{attribute addProperty BoxType "BK1250-0000-0017"}
{attribute addProperty Id "Term_387_KL1002KL1002_D229A9CA00"}
{attribute addProperty CRC "1147850243"}
{attribute addProperty SizeInBites "0"}
{attribute addProperty SizeInBytes "0"}
TYPE A_0016_BK1250_0000_0017_446ACE03 EXTENDS BK1250_4487A81F :
STRUCT
	{attribute addProperty Name "Term_387_KL1002"}
	Term_387_KL1002 : KL1002_D229A9CA;
END_STRUCT
END_TYPE

(* stored: Version 1.2.0.0, ProductVersion 3.1.4024.9
   DUT A_0016_BK1250_0000_0017_446ACE03: Id {7f26ba5c-4b3e-4757-8f86-78cc9b3a9382} *)
